INTERFACE IEventHandlerBase EXTENDS __SYSTEM.IQueryInterface

END_INTERFACE

(* stored: Version 1.1.0.1, ProductVersion 3.1.4024.3
   Itf IEventHandlerBase: Id {93405f16-7fa2-4417-ba8a-7d9a9d4c70ce} *)
